(* PLC project SafeLOGIC, BrAutomation SafeDESIGNER  5.24.1.0 *)
(* stored: companyURL http://www.br-automation.com, creationDateTime Sun Dec 07 16:37:42 2025 *)

PROGRAM VENTILATION
  VAR  (* added by the conversion: wires and edge detectors of the diagram *)
    _GE_S1247_OUT : SAFEDINT;
  END_VAR

(* FBD diagram, written out as Structured Text *)
(* FuB - Ventilation *)
(* Function 09 - Customer room ventilation *)
(* Alarm *)
(* Safety loop *)
(* Muting --> GCB ON + 10s *)
xET_TOF1(IN := OR_S(sDI_ERV_Cust, NOT_S(sbGCB_On_10s)), PT := SAFETIME#15s);
xDI_MON_ERV_Cust(sDI := xET_TOF1.Q, sbPara_Exist := PARA_ERV_Cust_Active, sbSafeInputOK := sbSafeInputOK_ERV_Cust);
bAMM_A9417 := xDI_MON_ERV_Cust.bAlarm;
(* Channel error *)
(* Warning *)
(* Elapsed time *)
iOUT_F09_Cust_OK_15s_ET := xET_TOF1.iOUT_ET;
bAMM_W9524 := xDI_MON_ERV_Cust.bWarning;
sbSL_OK_Cust := xDI_MON_ERV_Cust.sbSL_OK;
(* Plausibility check at standstill *)
(* Warning *)
(* Safety loop *)
xET1(IN := AND_S(sbN_Standstill, sDI_ERV_Cust), PT := SAFETIME#5h);
xKeepAMM_2s_W1(sbAMMxxxx := OR_S(NOT_S(PARA_ERV_Cust_Active), NOT_S(xET1.Q)));
bAMM_W9523 := xKeepAMM_2s_W1.bAMMxxxx;
sbSL_OK_Cust_PC := xKeepAMM_2s_W1.sbSL_OK;
(* Elapsed time *)
iOUT_F09_Cust_PC_ET := xET1.iOUT_ET;
(* Plausibility check OK *)
bOUT_F09_Cust_OK_PC := SAFEBOOL_TO_BOOL(AND_S(sbN_Standstill, NOT_S(sDI_ERV_Cust)));
(* HMI - Customer room ventilation is operating *)
(* Customer room ventilation in operation *)
bOUT_F09_Cust_OK := SAFEBOOL_TO_BOOL(OR_S(NOT_S(PARA_ERV_Cust_Active), AND_S(sbGCB_On_10s, sDI_ERV_Cust)));
(* Status of digital input *)
(* Customer room ventilation - Status of digital input *)
bOUT_F09_DI_ERV_Cust := SAFEBOOL_TO_BOOL(sDI_ERV_Cust);
(* Function 09 - Doors *)
(* Alarm *)
(* Muting --> GCB ON + 10s *)
(* Safety loop *)
xET_TOF2(IN := OR_S(sDI_ER_Door_CL, NOT_S(sbGCB_On_10s)), PT := SAFETIME#15s);
xDI_MON_ER_Door_CL(sDI := xET_TOF2.Q, sbPara_Exist := AND_S(PARA_ER_Door_MonActive, NOT_S(PARA_ERV_Cust_Active)), sbSafeInputOK := sbSafeInputOK_ER_Door_CL);
bAMM_A9480 := xDI_MON_ER_Door_CL.bAlarm;
sbSL_OK_Door_CL := xDI_MON_ER_Door_CL.sbSL_OK;
(* Warning *)
(* Channel error *)
(* Elapsed time *)
iOUT_F09_Door_OK_15s_ET := xET_TOF2.iOUT_ET;
bAMM_W9628 := xDI_MON_ER_Door_CL.bWarning;
(* Plausibility check at standstill *)
(* Warning *)
xTON1(IN := sDI_ER_Door_CL, PT := SAFETIME#24d);
xKeepAMM_2s_W2(sbAMMxxxx := OR_S(PARA_ERV_Cust_Active, NOT_S(PARA_ER_Door_MonActive), NOT_S(xTON1.Q)));
bAMM_W9627 := xKeepAMM_2s_W2.bAMMxxxx;
(* HMI - Engine room doors are closed *)
(* Engine room doors are closed *)
bOUT_F09_Door_OK := SAFEBOOL_TO_BOOL(OR_S(PARA_ERV_Cust_Active, NOT_S(PARA_ER_Door_MonActive), AND_S(sbGCB_On_10s, sDI_ER_Door_CL)));
(* Function 09 - Cold country mode *)
sbColdMode_Active := AND_S(PARA_ERV_ColdCountry_Active, BOOL_TO_SAFEBOOL(bIN_ERV_ColdCountry));
(* Function 09 - Fans *)
xERV_INL1_Fan(PARA_Fan_Active := AND_S(NOT_S(PARA_ERV_Cust_Active), GE_S(PARA_Nr_ERV_INL_Fan, SAFEDINT#1)), sbColdMode_Active := sbColdMode_Active, sbGCB_On_10s := sbGCB_On_10s, sbN_Standstill := sbN_Standstill, sDI_ERV_Fan_Run := sDI_ERV_INL1_Fan_Run, sbSafeInputOK_ERV_Fan_Run := sbSafeInputOK_ERV_INL1_Fan_Run);
bOUT_F09_INL1_Fan_OK := xERV_INL1_Fan.bOUT_Fan_OK;
bAMM_W9629 := xERV_INL1_Fan.bAMM_Fan;
bAMM_W9630 := xERV_INL1_Fan.bAMM_Fan_PC;
iOUT_F09_INL1_Fan_OK_1m_ET := xERV_INL1_Fan.iOUT_Fan_OK_1m_ET;
bOUT_F09_INL1_Fan_OK_PC := xERV_INL1_Fan.bOUT_Fan_OK_PC;
bAMM_W9631 := xERV_INL1_Fan.bAMM_Fan_NV;
sbSL_OK_INL1_Fan := xERV_INL1_Fan.sbSL_OK;
xERV_INL2_Fan(PARA_Fan_Active := AND_S(NOT_S(PARA_ERV_Cust_Active), GE_S(PARA_Nr_ERV_INL_Fan, SAFEDINT#2)), sbColdMode_Active := sbColdMode_Active, sbGCB_On_10s := sbGCB_On_10s, sbN_Standstill := sbN_Standstill, sDI_ERV_Fan_Run := sDI_ERV_INL2_Fan_Run, sbSafeInputOK_ERV_Fan_Run := sbSafeInputOK_ERV_INL2_Fan_Run);
bOUT_F09_INL2_Fan_OK := xERV_INL2_Fan.bOUT_Fan_OK;
bAMM_W9632 := xERV_INL2_Fan.bAMM_Fan;
bOUT_F09_INL2_Fan_OK_PC := xERV_INL2_Fan.bOUT_Fan_OK_PC;
bAMM_W9633 := xERV_INL2_Fan.bAMM_Fan_PC;
iOUT_F09_INL2_Fan_OK_1m_ET := xERV_INL2_Fan.iOUT_Fan_OK_1m_ET;
bAMM_W9634 := xERV_INL2_Fan.bAMM_Fan_NV;
sbSL_OK_INL2_Fan := xERV_INL2_Fan.sbSL_OK;
xERV_INL3_Fan(PARA_Fan_Active := AND_S(NOT_S(PARA_ERV_Cust_Active), GE_S(PARA_Nr_ERV_INL_Fan, SAFEDINT#3)), sbColdMode_Active := sbColdMode_Active, sbGCB_On_10s := sbGCB_On_10s, sbN_Standstill := sbN_Standstill, sDI_ERV_Fan_Run := sDI_ERV_INL3_Fan_Run, sbSafeInputOK_ERV_Fan_Run := sbSafeInputOK_ERV_INL3_Fan_Run);
bAMM_W9635 := xERV_INL3_Fan.bAMM_Fan;
bAMM_W9636 := xERV_INL3_Fan.bAMM_Fan_PC;
iOUT_F09_INL3_Fan_OK_1m_ET := xERV_INL3_Fan.iOUT_Fan_OK_1m_ET;
bOUT_F09_INL3_Fan_OK := xERV_INL3_Fan.bOUT_Fan_OK;
bOUT_F09_INL3_Fan_OK_PC := xERV_INL3_Fan.bOUT_Fan_OK_PC;
bAMM_W9637 := xERV_INL3_Fan.bAMM_Fan_NV;
sbSL_OK_INL3_Fan := xERV_INL3_Fan.sbSL_OK;
xERV_INL4_Fan(PARA_Fan_Active := AND_S(NOT_S(PARA_ERV_Cust_Active), GE_S(PARA_Nr_ERV_INL_Fan, SAFEDINT#4)), sbColdMode_Active := sbColdMode_Active, sbGCB_On_10s := sbGCB_On_10s, sbN_Standstill := sbN_Standstill, sDI_ERV_Fan_Run := sDI_ERV_INL4_Fan_Run, sbSafeInputOK_ERV_Fan_Run := sbSafeInputOK_ERV_INL4_Fan_Run);
bAMM_W9638 := xERV_INL4_Fan.bAMM_Fan;
bAMM_W9639 := xERV_INL4_Fan.bAMM_Fan_PC;
iOUT_F09_INL4_Fan_OK_1m_ET := xERV_INL4_Fan.iOUT_Fan_OK_1m_ET;
bOUT_F09_INL4_Fan_OK := xERV_INL4_Fan.bOUT_Fan_OK;
bOUT_F09_INL4_Fan_OK_PC := xERV_INL4_Fan.bOUT_Fan_OK_PC;
bAMM_W9640 := xERV_INL4_Fan.bAMM_Fan_NV;
sbSL_OK_INL4_Fan := xERV_INL4_Fan.sbSL_OK;
xERV_INL5_Fan(PARA_Fan_Active := AND_S(NOT_S(PARA_ERV_Cust_Active), GE_S(PARA_Nr_ERV_INL_Fan, SAFEDINT#5)), sbColdMode_Active := sbColdMode_Active, sbGCB_On_10s := sbGCB_On_10s, sbN_Standstill := sbN_Standstill, sDI_ERV_Fan_Run := sDI_ERV_INL5_Fan_Run, sbSafeInputOK_ERV_Fan_Run := sbSafeInputOK_ERV_INL5_Fan_Run);
bAMM_W9641 := xERV_INL5_Fan.bAMM_Fan;
bAMM_W9642 := xERV_INL5_Fan.bAMM_Fan_PC;
iOUT_F09_INL5_Fan_OK_1m_ET := xERV_INL5_Fan.iOUT_Fan_OK_1m_ET;
bOUT_F09_INL5_Fan_OK := xERV_INL5_Fan.bOUT_Fan_OK;
bOUT_F09_INL5_Fan_OK_PC := xERV_INL5_Fan.bOUT_Fan_OK_PC;
bAMM_W9643 := xERV_INL5_Fan.bAMM_Fan_NV;
sbSL_OK_INL5_Fan := xERV_INL5_Fan.sbSL_OK;
xERV_INL6_Fan(PARA_Fan_Active := AND_S(NOT_S(PARA_ERV_Cust_Active), EQ_S(PARA_Nr_ERV_INL_Fan, SAFEDINT#6)), sbColdMode_Active := sbColdMode_Active, sbGCB_On_10s := sbGCB_On_10s, sbN_Standstill := sbN_Standstill, sDI_ERV_Fan_Run := sDI_ERV_INL6_Fan_Run, sbSafeInputOK_ERV_Fan_Run := sbSafeInputOK_ERV_INL6_Fan_Run);
bAMM_W9644 := xERV_INL6_Fan.bAMM_Fan;
bAMM_W9645 := xERV_INL6_Fan.bAMM_Fan_PC;
iOUT_F09_INL6_Fan_OK_1m_ET := xERV_INL6_Fan.iOUT_Fan_OK_1m_ET;
bOUT_F09_INL6_Fan_OK := xERV_INL6_Fan.bOUT_Fan_OK;
bOUT_F09_INL6_Fan_OK_PC := xERV_INL6_Fan.bOUT_Fan_OK_PC;
bAMM_W9646 := xERV_INL6_Fan.bAMM_Fan_NV;
sbSL_OK_INL6_Fan := xERV_INL6_Fan.sbSL_OK;
xERV_NrFailed_Fan(PARA_Nr := PARA_Nr_ERV_INL_Fan, PARA_NrMaxErr := PARA_NrMaxErr_ERV_INL_Fan, sbSL_OK_Group1 := sbSL_OK_INL1_Fan, sbSL_OK_Group2 := sbSL_OK_INL2_Fan, sbSL_OK_Group3 := sbSL_OK_INL3_Fan, sbSL_OK_Group4 := sbSL_OK_INL4_Fan, sbSL_OK_Group5 := sbSL_OK_INL5_Fan, sbSL_OK_Group6 := sbSL_OK_INL6_Fan);
bAMM_A9481 := xERV_NrFailed_Fan.bAMM_NrMax;
sbSL_OK_INL_Fan_All := xERV_NrFailed_Fan.sbSL_OK_All;
(* Function 09 - Inlet louvres *)
xERV_INL1_Lou(PARA_Lou_Active := AND_S(NOT_S(PARA_ERV_Cust_Active), GE_S(PARA_Nr_ERV_INL_Lou, SAFEDINT#1)), sbColdMode_Active := sbColdMode_Active, sbN_Standstill := sbN_Standstill, sbGasValves_Closed := sbGasValves_Closed, sDI_ERV_Lou_OP := sDI_ERV_INL1_Lou_OP, sDI_ERV_Lou_CL := sDI_ERV_INL1_Lou_CL, sbSafeInputOK_ERV_Lou_OP := sbSafeInputOK_ERV_INL1_Lou_OP, sbSafeInputOK_ERV_Lou_CL := sbSafeInputOK_ERV_INL1_Lou_CL);
bOUT_F09_INL1_Lou_OK := xERV_INL1_Lou.bOUT_Lou_OK;
bAMM_W9647 := xERV_INL1_Lou.bAMM_Lou_OP;
bOUT_F09_INL1_Lou_OK_PC := xERV_INL1_Lou.bOUT_Lou_OK_PC;
bAMM_W9648 := xERV_INL1_Lou.bAMM_Lou_CL;
iOUT_F09_INL1_Lou_OK_1m_ET := xERV_INL1_Lou.iOUT_Lou_OK_1m_ET;
bAMM_W9649 := xERV_INL1_Lou.bAMM_Lou_OP_NV;
sbSL_OK_INL1_Lou := xERV_INL1_Lou.sbSL_OK;
bAMM_W9650 := xERV_INL1_Lou.bAMM_Lou_CL_NV;
bAMM_W9651 := xERV_INL1_Lou.bAMM_Lou_PC;
xERV_INL2_Lou(PARA_Lou_Active := AND_S(NOT_S(PARA_ERV_Cust_Active), GE_S(PARA_Nr_ERV_INL_Lou, SAFEDINT#2)), sbColdMode_Active := sbColdMode_Active, sbN_Standstill := sbN_Standstill, sbGasValves_Closed := sbGasValves_Closed, sDI_ERV_Lou_OP := sDI_ERV_INL2_Lou_OP, sDI_ERV_Lou_CL := sDI_ERV_INL2_Lou_CL, sbSafeInputOK_ERV_Lou_OP := sbSafeInputOK_ERV_INL2_Lou_OP, sbSafeInputOK_ERV_Lou_CL := sbSafeInputOK_ERV_INL2_Lou_CL);
bOUT_F09_INL2_Lou_OK := xERV_INL2_Lou.bOUT_Lou_OK;
bAMM_W9652 := xERV_INL2_Lou.bAMM_Lou_OP;
bOUT_F09_INL2_Lou_OK_PC := xERV_INL2_Lou.bOUT_Lou_OK_PC;
bAMM_W9653 := xERV_INL2_Lou.bAMM_Lou_CL;
iOUT_F09_INL2_Lou_OK_1m_ET := xERV_INL2_Lou.iOUT_Lou_OK_1m_ET;
bAMM_W9654 := xERV_INL2_Lou.bAMM_Lou_OP_NV;
sbSL_OK_INL2_Lou := xERV_INL2_Lou.sbSL_OK;
bAMM_W9655 := xERV_INL2_Lou.bAMM_Lou_CL_NV;
bAMM_W9656 := xERV_INL2_Lou.bAMM_Lou_PC;
xERV_INL3_Lou(PARA_Lou_Active := AND_S(NOT_S(PARA_ERV_Cust_Active), GE_S(PARA_Nr_ERV_INL_Lou, SAFEDINT#3)), sbColdMode_Active := sbColdMode_Active, sbN_Standstill := sbN_Standstill, sbGasValves_Closed := sbGasValves_Closed, sDI_ERV_Lou_OP := sDI_ERV_INL3_Lou_OP, sDI_ERV_Lou_CL := sDI_ERV_INL3_Lou_CL, sbSafeInputOK_ERV_Lou_OP := sbSafeInputOK_ERV_INL3_Lou_OP, sbSafeInputOK_ERV_Lou_CL := sbSafeInputOK_ERV_INL3_Lou_CL);
bOUT_F09_INL3_Lou_OK := xERV_INL3_Lou.bOUT_Lou_OK;
bAMM_W9657 := xERV_INL3_Lou.bAMM_Lou_OP;
bOUT_F09_INL3_Lou_OK_PC := xERV_INL3_Lou.bOUT_Lou_OK_PC;
bAMM_W9658 := xERV_INL3_Lou.bAMM_Lou_CL;
iOUT_F09_INL3_Lou_OK_1m_ET := xERV_INL3_Lou.iOUT_Lou_OK_1m_ET;
bAMM_W9659 := xERV_INL3_Lou.bAMM_Lou_OP_NV;
sbSL_OK_INL3_Lou := xERV_INL3_Lou.sbSL_OK;
bAMM_W9660 := xERV_INL3_Lou.bAMM_Lou_CL_NV;
bAMM_W9661 := xERV_INL3_Lou.bAMM_Lou_PC;
xERV_INL4_Lou(PARA_Lou_Active := AND_S(NOT_S(PARA_ERV_Cust_Active), GE_S(PARA_Nr_ERV_INL_Lou, SAFEDINT#4)), sbColdMode_Active := sbColdMode_Active, sbN_Standstill := sbN_Standstill, sbGasValves_Closed := sbGasValves_Closed, sDI_ERV_Lou_OP := sDI_ERV_INL4_Lou_OP, sDI_ERV_Lou_CL := sDI_ERV_INL4_Lou_CL, sbSafeInputOK_ERV_Lou_OP := sbSafeInputOK_ERV_INL4_Lou_OP, sbSafeInputOK_ERV_Lou_CL := sbSafeInputOK_ERV_INL4_Lou_CL);
bOUT_F09_INL4_Lou_OK := xERV_INL4_Lou.bOUT_Lou_OK;
bAMM_W9662 := xERV_INL4_Lou.bAMM_Lou_OP;
bOUT_F09_INL4_Lou_OK_PC := xERV_INL4_Lou.bOUT_Lou_OK_PC;
bAMM_W9663 := xERV_INL4_Lou.bAMM_Lou_CL;
iOUT_F09_INL4_Lou_OK_1m_ET := xERV_INL4_Lou.iOUT_Lou_OK_1m_ET;
bAMM_W9664 := xERV_INL4_Lou.bAMM_Lou_OP_NV;
sbSL_OK_INL4_Lou := xERV_INL4_Lou.sbSL_OK;
bAMM_W9665 := xERV_INL4_Lou.bAMM_Lou_CL_NV;
bAMM_W9666 := xERV_INL4_Lou.bAMM_Lou_PC;
xERV_INL5_Lou(PARA_Lou_Active := AND_S(NOT_S(PARA_ERV_Cust_Active), GE_S(PARA_Nr_ERV_INL_Lou, SAFEDINT#5)), sbColdMode_Active := sbColdMode_Active, sbN_Standstill := sbN_Standstill, sbGasValves_Closed := sbGasValves_Closed, sDI_ERV_Lou_OP := sDI_ERV_INL5_Lou_OP, sDI_ERV_Lou_CL := sDI_ERV_INL5_Lou_CL, sbSafeInputOK_ERV_Lou_OP := sbSafeInputOK_ERV_INL5_Lou_OP, sbSafeInputOK_ERV_Lou_CL := sbSafeInputOK_ERV_INL5_Lou_CL);
bOUT_F09_INL5_Lou_OK := xERV_INL5_Lou.bOUT_Lou_OK;
bAMM_W9667 := xERV_INL5_Lou.bAMM_Lou_OP;
bOUT_F09_INL5_Lou_OK_PC := xERV_INL5_Lou.bOUT_Lou_OK_PC;
bAMM_W9668 := xERV_INL5_Lou.bAMM_Lou_CL;
iOUT_F09_INL5_Lou_OK_1m_ET := xERV_INL5_Lou.iOUT_Lou_OK_1m_ET;
bAMM_W9669 := xERV_INL5_Lou.bAMM_Lou_OP_NV;
sbSL_OK_INL5_Lou := xERV_INL5_Lou.sbSL_OK;
bAMM_W9670 := xERV_INL5_Lou.bAMM_Lou_CL_NV;
bAMM_W9671 := xERV_INL5_Lou.bAMM_Lou_PC;
xERV_INL6_Lou(PARA_Lou_Active := AND_S(NOT_S(PARA_ERV_Cust_Active), EQ_S(PARA_Nr_ERV_INL_Lou, SAFEDINT#6)), sbColdMode_Active := sbColdMode_Active, sbN_Standstill := sbN_Standstill, sbGasValves_Closed := sbGasValves_Closed, sDI_ERV_Lou_OP := sDI_ERV_INL6_Lou_OP, sDI_ERV_Lou_CL := sDI_ERV_INL6_Lou_CL, sbSafeInputOK_ERV_Lou_OP := sbSafeInputOK_ERV_INL6_Lou_OP, sbSafeInputOK_ERV_Lou_CL := sbSafeInputOK_ERV_INL6_Lou_CL);
bOUT_F09_INL6_Lou_OK := xERV_INL6_Lou.bOUT_Lou_OK;
bAMM_W9672 := xERV_INL6_Lou.bAMM_Lou_OP;
bOUT_F09_INL6_Lou_OK_PC := xERV_INL6_Lou.bOUT_Lou_OK_PC;
bAMM_W9673 := xERV_INL6_Lou.bAMM_Lou_CL;
iOUT_F09_INL6_Lou_OK_1m_ET := xERV_INL6_Lou.iOUT_Lou_OK_1m_ET;
bAMM_W9674 := xERV_INL6_Lou.bAMM_Lou_OP_NV;
sbSL_OK_INL6_Lou := xERV_INL6_Lou.sbSL_OK;
bAMM_W9675 := xERV_INL6_Lou.bAMM_Lou_CL_NV;
bAMM_W9676 := xERV_INL6_Lou.bAMM_Lou_PC;
xERV_NrFailed_INL_Lou(PARA_Nr := PARA_Nr_ERV_INL_Lou, PARA_NrMaxErr := PARA_NrMaxErr_ERV_INL_Lou, sbSL_OK_Group1 := sbSL_OK_INL1_Lou, sbSL_OK_Group2 := sbSL_OK_INL2_Lou, sbSL_OK_Group3 := sbSL_OK_INL3_Lou, sbSL_OK_Group4 := sbSL_OK_INL4_Lou, sbSL_OK_Group5 := sbSL_OK_INL5_Lou, sbSL_OK_Group6 := sbSL_OK_INL6_Lou);
bAMM_A9482 := xERV_NrFailed_INL_Lou.bAMM_NrMax;
sbSL_OK_INL_Lou_All := xERV_NrFailed_INL_Lou.sbSL_OK_All;
(* Function 09 - Outlet louvres *)
xERV_OTL1_Lou(PARA_Lou_Active := AND_S(NOT_S(PARA_ERV_Cust_Active), GE_S(PARA_Nr_ERV_OTL_Lou, SAFEDINT#1)), sbColdMode_Active := SAFEFALSE, sbN_Standstill := sbN_Standstill, sbGasValves_Closed := sbGasValves_Closed, sDI_ERV_Lou_OP := sDI_ERV_OTL1_Lou_OP, sDI_ERV_Lou_CL := sDI_ERV_OTL1_Lou_CL, sbSafeInputOK_ERV_Lou_OP := sbSafeInputOK_ERV_OTL1_Lou_OP, sbSafeInputOK_ERV_Lou_CL := sbSafeInputOK_ERV_OTL1_Lou_CL);
bOUT_F09_OTL1_Lou_OK := xERV_OTL1_Lou.bOUT_Lou_OK;
bOUT_F09_OTL1_Lou_OK_PC := xERV_OTL1_Lou.bOUT_Lou_OK_PC;
bAMM_W9677 := xERV_OTL1_Lou.bAMM_Lou_CL;
iOUT_F09_OTL1_Lou_OK_1m_ET := xERV_OTL1_Lou.iOUT_Lou_OK_1m_ET;
bAMM_W9678 := xERV_OTL1_Lou.bAMM_Lou_OP_NV;
sbSL_OK_OTL1_Lou := xERV_OTL1_Lou.sbSL_OK;
bAMM_W9679 := xERV_OTL1_Lou.bAMM_Lou_CL_NV;
bAMM_W9680 := xERV_OTL1_Lou.bAMM_Lou_PC;
xERV_OTL2_Lou(PARA_Lou_Active := AND_S(NOT_S(PARA_ERV_Cust_Active), GE_S(PARA_Nr_ERV_OTL_Lou, SAFEDINT#2)), sbColdMode_Active := SAFEFALSE, sbN_Standstill := sbN_Standstill, sbGasValves_Closed := sbGasValves_Closed, sDI_ERV_Lou_OP := sDI_ERV_OTL2_Lou_OP, sDI_ERV_Lou_CL := sDI_ERV_OTL2_Lou_CL, sbSafeInputOK_ERV_Lou_OP := sbSafeInputOK_ERV_OTL2_Lou_OP, sbSafeInputOK_ERV_Lou_CL := sbSafeInputOK_ERV_OTL2_Lou_CL);
bOUT_F09_OTL2_Lou_OK := xERV_OTL2_Lou.bOUT_Lou_OK;
bOUT_F09_OTL2_Lou_OK_PC := xERV_OTL2_Lou.bOUT_Lou_OK_PC;
bAMM_W9681 := xERV_OTL2_Lou.bAMM_Lou_CL;
iOUT_F09_OTL2_Lou_OK_1m_ET := xERV_OTL2_Lou.iOUT_Lou_OK_1m_ET;
bAMM_W9682 := xERV_OTL2_Lou.bAMM_Lou_OP_NV;
sbSL_OK_OTL2_Lou := xERV_OTL2_Lou.sbSL_OK;
bAMM_W9683 := xERV_OTL2_Lou.bAMM_Lou_CL_NV;
bAMM_W9684 := xERV_OTL2_Lou.bAMM_Lou_PC;
xERV_OTL3_Lou(PARA_Lou_Active := AND_S(NOT_S(PARA_ERV_Cust_Active), GE_S(PARA_Nr_ERV_OTL_Lou, SAFEDINT#3)), sbColdMode_Active := SAFEFALSE, sbN_Standstill := sbN_Standstill, sbGasValves_Closed := sbGasValves_Closed, sDI_ERV_Lou_OP := sDI_ERV_OTL3_Lou_OP, sDI_ERV_Lou_CL := sDI_ERV_OTL3_Lou_CL, sbSafeInputOK_ERV_Lou_OP := sbSafeInputOK_ERV_OTL3_Lou_OP, sbSafeInputOK_ERV_Lou_CL := sbSafeInputOK_ERV_OTL3_Lou_CL);
bOUT_F09_OTL3_Lou_OK := xERV_OTL3_Lou.bOUT_Lou_OK;
bOUT_F09_OTL3_Lou_OK_PC := xERV_OTL3_Lou.bOUT_Lou_OK_PC;
bAMM_W9685 := xERV_OTL3_Lou.bAMM_Lou_CL;
iOUT_F09_OTL3_Lou_OK_1m_ET := xERV_OTL3_Lou.iOUT_Lou_OK_1m_ET;
bAMM_W9686 := xERV_OTL3_Lou.bAMM_Lou_OP_NV;
sbSL_OK_OTL3_Lou := xERV_OTL3_Lou.sbSL_OK;
bAMM_W9687 := xERV_OTL3_Lou.bAMM_Lou_CL_NV;
bAMM_W9688 := xERV_OTL3_Lou.bAMM_Lou_PC;
xERV_OTL4_Lou(PARA_Lou_Active := AND_S(NOT_S(PARA_ERV_Cust_Active), GE_S(PARA_Nr_ERV_OTL_Lou, SAFEDINT#4)), sbColdMode_Active := SAFEFALSE, sbN_Standstill := sbN_Standstill, sbGasValves_Closed := sbGasValves_Closed, sDI_ERV_Lou_OP := sDI_ERV_OTL4_Lou_OP, sDI_ERV_Lou_CL := sDI_ERV_OTL4_Lou_CL, sbSafeInputOK_ERV_Lou_OP := sbSafeInputOK_ERV_OTL4_Lou_OP, sbSafeInputOK_ERV_Lou_CL := sbSafeInputOK_ERV_OTL4_Lou_CL);
bOUT_F09_OTL4_Lou_OK := xERV_OTL4_Lou.bOUT_Lou_OK;
bOUT_F09_OTL4_Lou_OK_PC := xERV_OTL4_Lou.bOUT_Lou_OK_PC;
bAMM_W9689 := xERV_OTL4_Lou.bAMM_Lou_CL;
iOUT_F09_OTL4_Lou_OK_1m_ET := xERV_OTL4_Lou.iOUT_Lou_OK_1m_ET;
bAMM_W9690 := xERV_OTL4_Lou.bAMM_Lou_OP_NV;
sbSL_OK_OTL4_Lou := xERV_OTL4_Lou.sbSL_OK;
bAMM_W9691 := xERV_OTL4_Lou.bAMM_Lou_CL_NV;
bAMM_W9692 := xERV_OTL4_Lou.bAMM_Lou_PC;
xERV_OTL5_Lou(PARA_Lou_Active := AND_S(NOT_S(PARA_ERV_Cust_Active), GE_S(PARA_Nr_ERV_OTL_Lou, SAFEDINT#5)), sbColdMode_Active := SAFEFALSE, sbN_Standstill := sbN_Standstill, sbGasValves_Closed := sbGasValves_Closed, sDI_ERV_Lou_OP := sDI_ERV_OTL5_Lou_OP, sDI_ERV_Lou_CL := sDI_ERV_OTL5_Lou_CL, sbSafeInputOK_ERV_Lou_OP := sbSafeInputOK_ERV_OTL5_Lou_OP, sbSafeInputOK_ERV_Lou_CL := sbSafeInputOK_ERV_OTL5_Lou_CL);
bOUT_F09_OTL5_Lou_OK := xERV_OTL5_Lou.bOUT_Lou_OK;
bOUT_F09_OTL5_Lou_OK_PC := xERV_OTL5_Lou.bOUT_Lou_OK_PC;
bAMM_W9693 := xERV_OTL5_Lou.bAMM_Lou_CL;
iOUT_F09_OTL5_Lou_OK_1m_ET := xERV_OTL5_Lou.iOUT_Lou_OK_1m_ET;
bAMM_W9694 := xERV_OTL5_Lou.bAMM_Lou_OP_NV;
sbSL_OK_OTL5_Lou := xERV_OTL5_Lou.sbSL_OK;
bAMM_W9695 := xERV_OTL5_Lou.bAMM_Lou_CL_NV;
bAMM_W9696 := xERV_OTL5_Lou.bAMM_Lou_PC;
xERV_OTL6_Lou(PARA_Lou_Active := AND_S(NOT_S(PARA_ERV_Cust_Active), EQ_S(PARA_Nr_ERV_OTL_Lou, SAFEDINT#6)), sbColdMode_Active := SAFEFALSE, sbN_Standstill := sbN_Standstill, sbGasValves_Closed := sbGasValves_Closed, sDI_ERV_Lou_OP := sDI_ERV_OTL6_Lou_OP, sDI_ERV_Lou_CL := sDI_ERV_OTL6_Lou_CL, sbSafeInputOK_ERV_Lou_OP := sbSafeInputOK_ERV_OTL6_Lou_OP, sbSafeInputOK_ERV_Lou_CL := sbSafeInputOK_ERV_OTL6_Lou_CL);
bOUT_F09_OTL6_Lou_OK := xERV_OTL6_Lou.bOUT_Lou_OK;
bOUT_F09_OTL6_Lou_OK_PC := xERV_OTL6_Lou.bOUT_Lou_OK_PC;
bAMM_W9697 := xERV_OTL6_Lou.bAMM_Lou_CL;
iOUT_F09_OTL6_Lou_OK_1m_ET := xERV_OTL6_Lou.iOUT_Lou_OK_1m_ET;
bAMM_W9698 := xERV_OTL6_Lou.bAMM_Lou_OP_NV;
sbSL_OK_OTL6_Lou := xERV_OTL6_Lou.sbSL_OK;
bAMM_W9699 := xERV_OTL6_Lou.bAMM_Lou_CL_NV;
bAMM_W9700 := xERV_OTL6_Lou.bAMM_Lou_PC;
xERV_NrFailed_OTL_Lou(PARA_Nr := PARA_Nr_ERV_OTL_Lou, PARA_NrMaxErr := PARA_NrMaxErr_ERV_OTL_Lou, sbSL_OK_Group1 := sbSL_OK_OTL1_Lou, sbSL_OK_Group2 := sbSL_OK_OTL2_Lou, sbSL_OK_Group3 := sbSL_OK_OTL3_Lou, sbSL_OK_Group4 := sbSL_OK_OTL4_Lou, sbSL_OK_Group5 := sbSL_OK_OTL5_Lou, sbSL_OK_Group6 := sbSL_OK_OTL6_Lou);
bAMM_A9483 := xERV_NrFailed_OTL_Lou.bAMM_NrMax;
sbSL_OK_OTL_Lou_All := xERV_NrFailed_OTL_Lou.sbSL_OK_All;
(* Safety loop *)
sbF09_OK_Ventilation := AND_S(sbSL_OK_Cust, sbSL_OK_Cust_PC, sbSL_OK_Door_CL, sbSL_OK_INL_Fan_All, sbSL_OK_INL_Lou_All, sbSL_OK_OTL_Lou_All);
(* Number of plausibility checks not performed *)
xSF_RD(Activate := SAFEBOOL_TO_BOOL(NOT_S(PARA_ERV_Cust_Active)), S_DataID := iRD_Nr_PC_NotDone, S_DataIn := siNr_PC_NotDone_Save, S_DataInOK := SAFETRUE, S_Store := sbStore_Nr_PC_NotDone);
xR_TRIG(CLK := xSF_RD.S_DataOutOK);
xERV_PC_NotDone(PARA_Cust_Active := PARA_ERV_Cust_Active, sbN_Standstill := sbN_Standstill, bERV_Lou_PC_OP := bIN_ERV_Lou_PC_OP, bERV_Lou_PC_CL := bIN_ERV_Lou_PC_CL, siNr_PC_NotDone_Save := siNr_PC_NotDone_Save, siNr_PC_NotDone_Stored := xSF_RD.S_DataOut, sbNr_PC_ND_TakeOver := xR_TRIG.Q);
siNr_PC_NotDone := xERV_PC_NotDone.siNr_PC_NotDone;
(* Store counter remanent *)
sbStore_Nr_PC_NotDone := NOT_S(EQ_S(siNr_PC_NotDone, siNr_PC_NotDone_Save));
siNr_PC_NotDone_Save := siNr_PC_NotDone;
xSAFEDINT_TO_SAFEINT(IN := siNr_PC_NotDone);
iOUT_F09_Nr_PC_NotDone := SAFEINT_TO_INT(xSAFEDINT_TO_SAFEINT.OUT);
(* Forced plausibility check *)
_GE_S1247_OUT := GE_S(siNr_PC_NotDone, SAFEDINT#10);
bOUT_F09_ERV_PC_Forced := SAFEBOOL_TO_BOOL(_GE_S1247_OUT);
xKeepAMM_2s(sbAMMxxxx := OR_S(NOT_S(_GE_S1247_OUT), NOT_S(sbN_Standstill)));
bAMM_A9428 := xKeepAMM_2s.bAMMxxxx;
sbRel_GV_ERV_PC_OK := xKeepAMM_2s.sbSL_OK;
END_PROGRAM
